// TIA Portal V19 export
FUNCTION_BLOCK "Block_2"   // FB1, LAD
{ S7_Optimized_Access := 'TRUE' }
// stored: MemoryReserve 100, SetENOAutomatically false
   VAR_INPUT
      p : "pulsante";
   END_VAR
   VAR_OUTPUT
      L : Bool;
   END_VAR
BEGIN

REGION Network 1
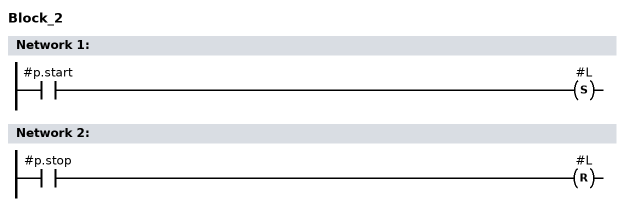
   RUNG wire#powerrail
      Contact( #p.start )
      S_Coil( #L )
   END_RUNG
   // the same network as SCL:
   IF #p.start THEN #L := TRUE; END_IF;
END_REGION

REGION Network 2
   RUNG wire#powerrail
      Contact( #p.stop )
      R_Coil( #L )
   END_RUNG
   // the same network as SCL:
   IF #p.stop THEN #L := FALSE; END_IF;
END_REGION
END_FUNCTION_BLOCK
